INTERFACE ITF_HighLevelSystem

PROPERTY eActivationStatus : ActivationStatus
GET
END_GET
SET
END_SET
END_PROPERTY

PROPERTY PUBLIC eCondition : HighLevelCondition
GET
END_GET
END_PROPERTY

PROPERTY PUBLIC nErrorID : UDINT
GET
END_GET
END_PROPERTY

END_INTERFACE

(* stored: Version 1.1.0.1, ProductVersion 3.1.4024.12
   Itf ITF_HighLevelSystem: Id {5dcd8f12-5bd1-43e6-9f2b-637a7956ae72}
   Property eActivationStatus: Id {f303fa50-e59e-47e2-b1a7-c5fd3df26395}
   Get Get: Id {fc4909dc-880e-45df-8875-4112267c9b9f}
   Set Set: Id {e10cb974-5a01-4e32-bd05-de3c2e892f39}
   Property eCondition: Id {d28282cf-876d-4d28-8a01-fb7919431854}
   Get Get: Id {97649c1c-a360-423a-85fe-e8e2a0f87e2b}
   Property nErrorID: Id {e9d4f733-cdaf-4ac8-b417-fe8362f4256b}
   Get Get: Id {6e161ed4-aa55-4cc2-81f1-ab9587af1fcb} *)
